Staubli VAL3: CheckPosEqual.pgx

program CheckPosEqual(pointRx x_pA (dimensions=1), bool& x_bPos (dimensions=1))
  local pointRx l_pHere
begin
  l_pHere=here(tTool,world)
  if power(x_pA.trsf.x-l_pHere.trsf.x,2)+power(x_pA.trsf.y-l_pHere.trsf.y,2)+power(x_pA.trsf.z-l_pHere.trsf.z,2)+power(x_pA.trsf.rx-l_pHere.trsf.rx,2)+power(x_pA.trsf.ry-l_pHere.trsf.ry,2)+power(x_pA.trsf.rz-l_pHere.trsf.rz,2)<0.2
    x_bPos=true
  else
    x_bPos=false
  endIf
end
